Staubli VAL3: link_it.pgx

public program link_it(string x_sName)
begin
  // link ALL
  call link_all(x_sName)
  // put the base config
  tTraj[x_sName].tData[0].tSuper.toStop=true
  tTraj[x_sName].tData[0].tSuper.moveType=1
  tTraj[x_sName].tData[0].tSuper.comment=""
  tTraj[x_sName].trAppro[0]={0,0,-50,0,0,0}
  tTraj[x_sName].trAppro[1]={0,0,-50,0,0,0}
  tTraj[x_sName].trDepart[0]={0,0,-50,0,0,0}
  tTraj[x_sName].trDepart[1]={0,0,-50,0,0,0}
end
